// Mitsubishi GX Works2 project: 인터록 회로   PLC: Q03UDV

PROGRAM MAIN
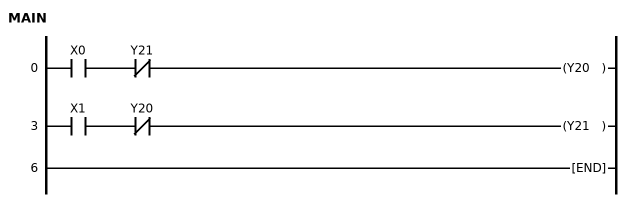
0     LD      X0
      ANI     Y21
      OUT     Y20
3     LD      X1
      ANI     Y20
      OUT     Y21
6     END
END_PROGRAM
